# EPICS autosave request: FOFBApp/Db/NDPluginBase_settings_mod.req
$(P)$(R)EnableCallbacks
$(P)$(R)MinCallbackTime
$(P)$(R)BlockingCallbacks
$(P)$(R)NDAttributesFile
